{library PUBLIC}
(* Use this function to close an open communication link to a specific device defined by Instance.
Returnvalue is true if closed ok otherwise false.*)
FUNCTION DeviceClose : BOOL
VAR_INPUT
	Instance: 				INT;		(* Instance is an address, use the function ToAddress() to convert station and device number to a valid address. *)
END_VAR

DeviceClose:=FALSE;
IF _GetInstance(Instance)=INSTANCE_STATUS.INSTANCE_STATUS_READY THEN
	IF _FreeInstance(Instance) THEN
		DeviceClose:=TRUE;
	END_IF;
END_IF;

END_FUNCTION

(* stored: Version 1.1.0.1, ProductVersion 3.1.4024.2
   POU DeviceClose: Id {2c3d7b64-3ac5-47b6-b093-7107eb16513b}, SpecialFunc None *)
